FUNCTION_BLOCK FB_SensorScaling
VAR_INPUT
	bExecute	: BOOL;
	iRawValue 	: INT;  //EL3058 raw meassure 16bits
	iSensorID	: INT;	//Sensor ID [1 for Festo | 2 for SMC Pressure Regulator]
END_VAR
VAR_OUTPUT
	bDone	 	: BOOL := FALSE; 
	rPressure 	: REAL; //Pressure output in Bar
END_VAR
VAR
	rScalingFactor : REAL;
    rOffset        : REAL;
END_VAR

//Scaling definition for each sensor
CASE iSensorID OF
    1:  //Festo MS6: 4-20mA → 0-6 bar
        rScalingFactor := 6.0 / (16384 - 3277);
        rOffset := -3277 * rScalingFactor;
		
    2:  //SMC ISE/ZSE20: 4-20mA → -0.100 to 1.000 MPa [1.0 a 10.0 bar]
        rScalingFactor := 11.0 / (16384 - 3277); //11 Bar Range
        rOffset := -1.0; 						 //Starts at -1.0 Bar
    ELSE
        rScalingFactor := 1.0;
        rOffset := 0.0;
END_CASE


//Applying the scaling
IF bExecute AND NOT bDone THEN
	rPressure 	:= rScalingFactor * TO_REAL(iRawValue) + rOffset;
	bDone		:= TRUE;
END_IF

END_FUNCTION_BLOCK

(* stored: Version 1.1.0.1, ProductVersion 3.1.4024.12
   POU FB_SensorScaling: Id {4c42e66e-2850-49c6-949b-9e520b1e950a}, SpecialFunc None *)
